FUNCTION_BLOCK FB_Obj_IOSchlauch
VAR_INPUT
	 
	I_bFrgNachladen				: BOOL;	(* Schrauber -> *)
	I_bVereinzelungskontrolle	: BOOL;	(* Schrauber -> *)
	I_bSotiertopfEin				: BOOL;	(* Schrauber -> *)

	I_bSchrauberBelegt			: BOOL;	(* Rütteltopf -> *)
	I_bSchlauchBelegt				: BOOL;	(* Rütteltopf -> *)
	I_bSchrAuswurfStart			: BOOL;	(* Rütteltopf -> *)

	I_bTasteVereinzelung			: BOOL;	(*am Rütteltopf*)
	I_bTasteNachruetteln			: BOOL;

	I_bNachladenaktiv 			: BOOL := FALSE;

END_VAR
VAR_OUTPUT
END_VAR
VAR
END_VAR

;

END_FUNCTION_BLOCK

(* stored: Version 1.1.0.1, ProductVersion 3.1.4024.3
   POU FB_Obj_IOSchlauch: Id {71dd367f-9899-4c52-8ea7-220b9a5d41b8}, SpecialFunc None *)
